# EPICS substitutions: iocs/fzoomExample/fzoomExampleApp/Db/fzoomExample.substitutions
file $(FZOOM)/db/fzoomStatus.template
{
    pattern {P, R, PORT, SCAN}
    {XF:16IDC, "{FZOOM}", FZOOM0, "10 second"}
}
file $(FZOOM)/db/fzoomCommand.template
{
    pattern {P, R, PORT}
    {XF:16IDC, "{FZOOM}", FZOOM0 }
}
